# EPICS substitutions: iocBoot/ioc14bmc/iocEnvVar.substitutions
#==============================================================================
#
# Abs:  IOC Administration Records
#
# Name: iocAdmin.substitutions
#
#==============================================================================
# Edited to work at BioCARS.

file "$(DEVIOCSTATS)/db/iocEnvVar.db"
{
pattern { IOCNAME, ENVNAME      , ENVVAR                          , ENVTYPE}
	{ 14BMC , LOCATION     , LOCATION                        , env    }
	{ 14BMC , ENGINEER     , ENGINEER                        , env    }
	{ 14BMC , CA_ADDR_LIST , EPICS_CA_ADDR_LIST              , epics  }
	{ 14BMC , CA_CONN_TIME , EPICS_CA_CONN_TMO               , epics  }
	{ 14BMC , CA_AUTO_ADDR , EPICS_CA_AUTO_ADDR_LIST         , epics  }
	{ 14BMC , CA_RPTR_PORT , EPICS_CA_REPEATER_PORT          , epics  }
	{ 14BMC , CA_SRVR_PORT , EPICS_CA_SERVER_PORT            , epics  }
	{ 14BMC , CA_MAX_ARRAY , EPICS_CA_MAX_ARRAY_BYTES        , epics  }
	{ 14BMC , CA_SRCH_TIME , EPICS_CA_MAX_SEARCH_PERIOD      , epics  }
	{ 14BMC , CA_BEAC_TIME , EPICS_CA_BEACON_PERIOD          , epics  }
	{ 14BMC , TIMEZONE     , EPICS_TIMEZONE                  , epics  }
	{ 14BMC , TS_NTP_INET  , EPICS_TS_NTP_INET               , epics  }
	{ 14BMC , IOC_LOG_PORT , EPICS_IOC_LOG_PORT              , epics  }
	{ 14BMC , IOC_LOG_INET , EPICS_IOC_LOG_INET              , epics  }
}
